FUNCTION_BLOCK ESP32_Testboard_12_DO (* Service Interface Function Block Type *)
  (* Function: All Outputs; Description: Copyright (c) 2018, 2023 Jose Cabral, HR Agrartechnik GmbH This program and the accompanying materials are made available under the terms of the Eclipse Public License 2.0 which is available at https://www.eclipse.org/legal/epl-2.0/ SPDX-License-Identifier: EPL-2.0 this maps to QX *)
  (* Version 1.0, 2018-12-05, Jose Cabral *)
  (* Version 1.1, 2022-08-04, Franz Höpfinger, HR Agrartechnik GmbH *)
  (* Version 1.2, 2023-01-05, Franz Höpfinger, HR Agrartechnik GmbH *)
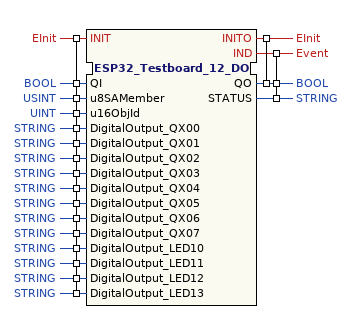
  EVENT_INPUT
    INIT : EInit WITH QI, u8SAMember, u16ObjId, DigitalOutput_QX00, DigitalOutput_QX01, DigitalOutput_QX02, DigitalOutput_QX03, DigitalOutput_QX04, DigitalOutput_QX05, DigitalOutput_QX06, DigitalOutput_QX07, DigitalOutput_LED10, DigitalOutput_LED11, DigitalOutput_LED12, DigitalOutput_LED13; (* Service Initialization *)
  END_EVENT
  EVENT_OUTPUT
    INITO : EInit WITH QO; (* Initialization Confirm *)
    IND WITH QO, STATUS; (* Indication from Resource *)
  END_EVENT
  VAR_INPUT
    QI : BOOL; (* Event Input Qualifier *)
    u8SAMember : USINT := GLOBAL; (* Dummy !, set to GLOBAL if in doubt. OFF deactivates FB. *)
    u16ObjId : UINT := ID_NULL; (* Dummy ! set to ID_NULL if in Doubt. ID_OFF deactivates FB. *)
    DigitalOutput_QX00 : STRING;
    DigitalOutput_QX01 : STRING;
    DigitalOutput_QX02 : STRING;
    DigitalOutput_QX03 : STRING;
    DigitalOutput_QX04 : STRING;
    DigitalOutput_QX05 : STRING;
    DigitalOutput_QX06 : STRING;
    DigitalOutput_QX07 : STRING;
    DigitalOutput_LED10 : STRING;
    DigitalOutput_LED11 : STRING;
    DigitalOutput_LED12 : STRING;
    DigitalOutput_LED13 : STRING;
  END_VAR
  VAR_OUTPUT
    QO : BOOL; (* Event Output Qualifier *)
    STATUS : STRING; (* Service Status *)
  END_VAR
END_FUNCTION_BLOCK
